// TIA Portal V19 export
FUNCTION "Digital_OUT" : Void   // FC2, LAD
{ S7_Optimized_Access := 'TRUE' }
// stored: SetENOAutomatically false
BEGIN

REGION Network 1: CMD Open IBC Valve
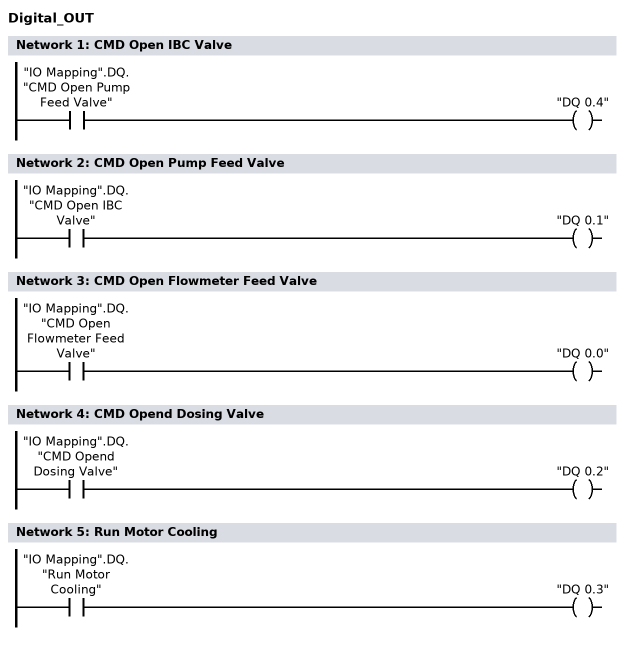
   RUNG wire#powerrail
      Contact( "IO Mapping".DQ."CMD Open Pump Feed Valve" )
      Coil( "DQ 0.4" )
   END_RUNG
   // the same network as SCL:
   "DQ 0.4" := "IO Mapping".DQ."CMD Open Pump Feed Valve";
END_REGION

REGION Network 2: CMD Open Pump Feed Valve
   RUNG wire#powerrail
      Contact( "IO Mapping".DQ."CMD Open IBC Valve" )
      Coil( "DQ 0.1" )
   END_RUNG
   // the same network as SCL:
   "DQ 0.1" := "IO Mapping".DQ."CMD Open IBC Valve";
END_REGION

REGION Network 3: CMD Open Flowmeter Feed Valve
   RUNG wire#powerrail
      Contact( "IO Mapping".DQ."CMD Open Flowmeter Feed Valve" )
      Coil( "DQ 0.0" )
   END_RUNG
   // the same network as SCL:
   "DQ 0.0" := "IO Mapping".DQ."CMD Open Flowmeter Feed Valve";
END_REGION

REGION Network 4: CMD Opend Dosing Valve
   RUNG wire#powerrail
      Contact( "IO Mapping".DQ."CMD Opend Dosing Valve" )
      Coil( "DQ 0.2" )
   END_RUNG
   // the same network as SCL:
   "DQ 0.2" := "IO Mapping".DQ."CMD Opend Dosing Valve";
END_REGION

REGION Network 5: Run Motor Cooling
   RUNG wire#powerrail
      Contact( "IO Mapping".DQ."Run Motor Cooling" )
      Coil( "DQ 0.3" )
   END_RUNG
   // the same network as SCL:
   "DQ 0.3" := "IO Mapping".DQ."Run Motor Cooling";
END_REGION
END_FUNCTION
